FUNCTION F_RealIsNaN : BOOL
VAR_INPUT
	rInput			: REAL;
END_VAR
VAR
	iBitWord		: DWORD;
	
	iExponent		: DWORD;
	iExponentMask	: DWORD := 2#0111_1111__1000_0000__0000_0000__0000_0000;
	
	iMantissa		: DWORD := 2#0000_0000__0111_1111__1111_1111__1111_1111;
	iMantissaMask	: DWORD := 2#0000_0000__0111_1111__1111_1111__1111_1111;
END_VAR

MEMCPY(ADR(iBitWord), ADR(rInput), SIZEOF(iBitWord));

iExponent	:= iBitWord AND iExponentMask;

iMantissa	:= iBitWord AND iMantissaMask;

IF iExponent = iExponentMask AND iMantissa <> 0 THEN
	F_RealIsNaN	:= TRUE;
ELSE
	F_RealIsNaN	:= FALSE;
END_IF

END_FUNCTION

(* stored: Version 1.1.0.1, ProductVersion 3.1.4024.12
   POU F_RealIsNaN: Id {f7e9610d-c963-4639-832a-2f4ef1c42da8}, SpecialFunc None *)
